FUNCTION Parameter2CellDataBlock : CellDataBlock
VAR_INPUT
	input : ParameterSet;
END_VAR
VAR
END_VAR

END_FUNCTION

(* stored: Version 1.1.0.1, ProductVersion 3.1.4022.10
   POU Parameter2CellDataBlock: Id {dd1c70da-073d-4d95-8332-934c34613ac4}, SpecialFunc None *)
